// TIA Portal V19 export
FUNCTION_BLOCK "LMG7ApcFr_Std"   // FB19206, LAD
{ S7_Optimized_Access := 'TRUE' }
// stored: AutoNumber false, MemoryReserve 100, SetENOAutomatically false
   VAR_INPUT
      FirstCycle : Bool;
      InterlockGeneral : Bool := TRUE;
      Reset : Bool;
      StepNumberStarted : Int := 2;
      Frequency_1s : Bool;
      DebugMode : Bool;
      ActualTime : Time_Of_Day;
   END_VAR
   VAR_OUTPUT
      ActiveStep : Int;
      StateStopped : Bool;
      StateStarting : Bool;
      StateStarted : Bool;
      StateStopping : Bool;
      StateError : Bool;
      State : Int;
      StepError : Int;
      HistoricBuffer : Struct
         Index : Int := 0;
         BufferDetail : Array[0..9] of Struct
            TimeStartStep : Time_Of_Day;
            StepNumber : Int;
            ElapseTime_s : Int;
         END_STRUCT;
      END_STRUCT;
   END_VAR
   VAR_IN_OUT
      StepRequested : Int;
      StepTimeOut : Int;
   END_VAR
   VAR
      statFrequency_1sOld : Bool;
      statEdgeUpFrequency_1s : Bool;
   END_VAR
   VAR RETAIN
      statStepRequested : Int;
      statCounterTimeOut : Int;
      StatHistoricBuffer : Struct
         Index : Int := 0;
         BufferDetail : Array[0..9] of Struct
            TimeStartStep : Time_Of_Day;
            StepNumber : Int;
            ElapseTime_s : Int;
         END_STRUCT;
      END_STRUCT;
   END_VAR
   VAR
      instF_TRIG_StepStopped { S7_SetPoint := 'True'} : F_TRIG;
      instF_TRIG_StepStarted { S7_SetPoint := 'True'} : F_TRIG;
   END_VAR
BEGIN

REGION Network 1 (SCL): (*** COMMENTS ***)
   //=============================================================================
   //SIEMENS AG
   //(c)Copyright 2016 All Rights Reserved
   //-----------------------------------------------------------------------------
   //Requirements:
   //Functionality: G7 management of step
   //               Hystoric buffer of 10 entries. Need egde of 1s and time of the PLC
   //Supported types:
   //-----------------------------------------------------------------------------
   //Change log table:
   //Version       Date            Expert in charge    Changes applied
   //01.01.00      09.04.2020      PdA                 First release
   //01.02.00      01.07.2021      PdA                 TimeOut management
   //                                                  New organization 
   //01.03.00      19.03.2024      PdA                 Replace Enable by FirstCycle
   //                                                  Delete InterlockStartUp parameters
   //=============================================================================
END_REGION

REGION Network 2 (SCL): First call
   IF #FirstCycle THEN
       #StateStopped := TRUE;
       #StateStarting := FALSE;
       #StateStarted := FALSE;
       #StateStopping := FALSE;
       #ActiveStep := 0;
       #StepTimeOut := 0;
       #StepRequested := 0;
       #StepError := 0;
       #statStepRequested := 0;
       #statCounterTimeOut := 0;
   END_IF;
END_REGION

REGION Network 3 (SCL): Step Requested
   IF NOT #StateError THEN
       IF NOT #InterlockGeneral THEN
           #statStepRequested := 0;
           #StepRequested := 0;
       ELSIF (#statCounterTimeOut > #StepTimeOut) THEN
           #statStepRequested := "LMAG7_STEP_NUMBER_ERROR";
           #StepError := #ActiveStep;
       ELSE
           #statStepRequested := #StepRequested;
       END_IF;
   ELSE
       IF #Reset THEN
           #statStepRequested := 0;
           #StepError := 0;
       END_IF;
   END_IF;

   IF (#statStepRequested <> #ActiveStep) THEN
       #ActiveStep := #statStepRequested;
       #StepRequested := #statStepRequested;

       #StatHistoricBuffer.Index := #StatHistoricBuffer.Index + 1;
       IF #StatHistoricBuffer.Index > 9 THEN
           #StatHistoricBuffer.Index := 0;
       END_IF;
       #StatHistoricBuffer.BufferDetail[#StatHistoricBuffer.Index].TimeStartStep := #ActualTime;
       #StatHistoricBuffer.BufferDetail[#StatHistoricBuffer.Index].StepNumber := #statStepRequested;
       #StatHistoricBuffer.BufferDetail[#StatHistoricBuffer.Index].ElapseTime_s := #statCounterTimeOut;

       #statCounterTimeOut := 0;
       #StepTimeOut := 0;

   END_IF;

   #statEdgeUpFrequency_1s := #Frequency_1s AND NOT #statFrequency_1sOld;
   #statFrequency_1sOld := #Frequency_1s;

   IF (#StepTimeOut > 0) AND #statEdgeUpFrequency_1s AND NOT #DebugMode THEN
       #statCounterTimeOut := #statCounterTimeOut + 1;
   END_IF;

   #ActiveStep := #statStepRequested;
END_REGION

REGION Network 4: Output State Stopped, Started, Error
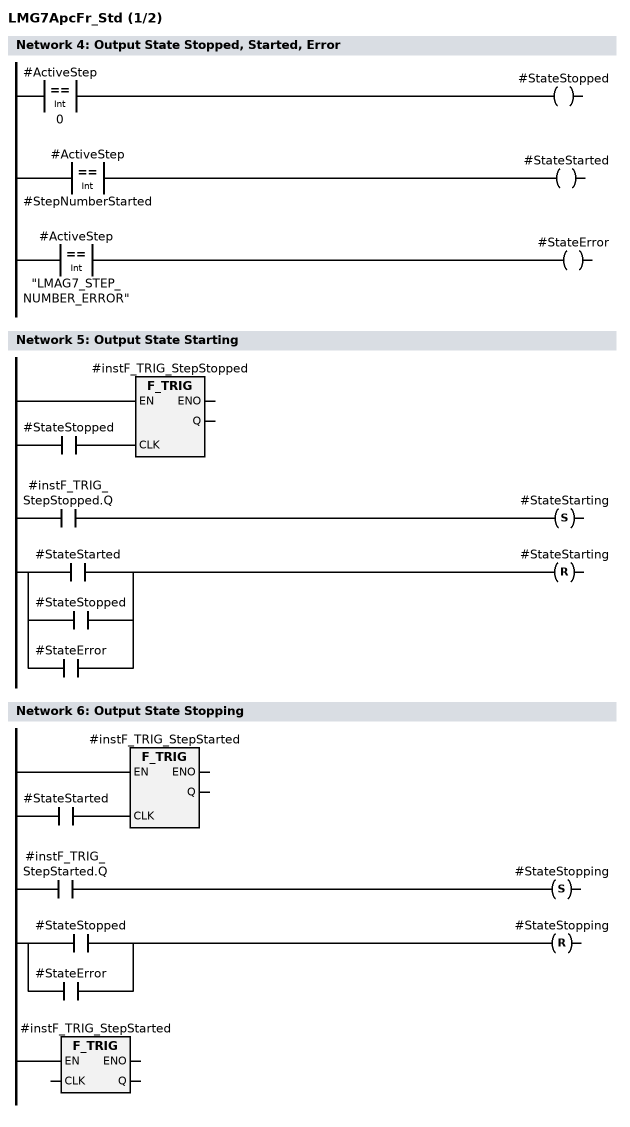
   RUNG wire#powerrail
      { S7_Templates := "SrcType := Int" } EQ_Contact(in1 := #ActiveStep, in2 := 0)
      Coil( #StateStopped )
   END_RUNG
   RUNG wire#powerrail
      { S7_Templates := "SrcType := Int" } EQ_Contact(in1 := #ActiveStep, in2 := #StepNumberStarted)
      Coil( #StateStarted )
   END_RUNG
   RUNG wire#powerrail
      { S7_Templates := "SrcType := Int" } EQ_Contact(in1 := #ActiveStep, in2 := "LMAG7_STEP_NUMBER_ERROR")
      Coil( #StateError )
   END_RUNG
   // the same network as SCL:
   #StateStopped := #ActiveStep = 0;
   #StateStarted := #ActiveStep = #StepNumberStarted;
   #StateError := #ActiveStep = "LMAG7_STEP_NUMBER_ERROR";
END_REGION

REGION Network 5: Output State Starting
   RUNG wire#powerrail
      #instF_TRIG_StepStopped.F_TRIG(CLK := wire#w1, Q =>)
   END_RUNG
   RUNG wire#powerrail
      Contact( #StateStopped )
   END_RUNG wire#w1
   RUNG wire#powerrail
      Contact( #instF_TRIG_StepStopped.Q )
      S_Coil( #StateStarting )
   END_RUNG
   RUNG wire#powerrail
      Contact( #StateStarted )
      wire#w2
      R_Coil( #StateStarting )
   END_RUNG
   RUNG wire#powerrail
      Contact( #StateStopped )
   END_RUNG wire#w2
   RUNG wire#powerrail
      Contact( #StateError )
   END_RUNG wire#w2
   // the same network as SCL:
   #instF_TRIG_StepStopped(CLK := #StateStopped);   // F_TRIG
   IF #instF_TRIG_StepStopped.Q THEN #StateStarting := TRUE; END_IF;
   IF #StateStarted OR #StateStopped OR #StateError THEN #StateStarting := FALSE; END_IF;
END_REGION

REGION Network 6: Output State Stopping
   RUNG wire#powerrail
      #instF_TRIG_StepStarted.F_TRIG(CLK := wire#w1, Q =>)
   END_RUNG
   RUNG wire#powerrail
      Contact( #StateStarted )
   END_RUNG wire#w1
   RUNG wire#powerrail
      Contact( #instF_TRIG_StepStarted.Q )
      S_Coil( #StateStopping )
   END_RUNG
   RUNG wire#powerrail
      Contact( #StateStopped )
      wire#w2
      R_Coil( #StateStopping )
   END_RUNG
   RUNG wire#powerrail
      Contact( #StateError )
   END_RUNG wire#w2
   RUNG wire#powerrail
      #instF_TRIG_StepStarted.F_TRIG(CLK :=, Q =>)
   END_RUNG
   // the same network as SCL:
   #instF_TRIG_StepStarted(CLK := #StateStarted);   // F_TRIG
   IF #instF_TRIG_StepStarted.Q THEN #StateStopping := TRUE; END_IF;
   IF #StateStopped OR #StateError THEN #StateStopping := FALSE; END_IF;
   #instF_TRIG_StepStarted();   // F_TRIG
END_REGION

REGION Network 7: Output State G7
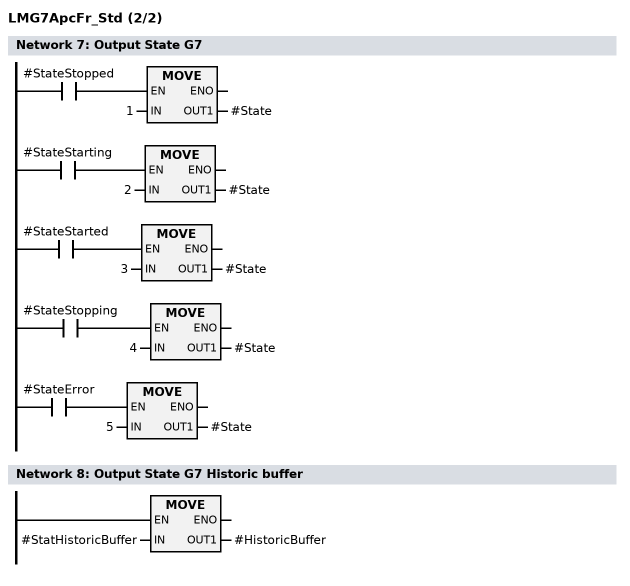
   RUNG wire#powerrail
      Contact( #StateStopped )
      Move(in := 1, out1 => #State)
   END_RUNG
   RUNG wire#powerrail
      Contact( #StateStarting )
      Move(in := 2, out1 => #State)
   END_RUNG
   RUNG wire#powerrail
      Contact( #StateStarted )
      Move(in := 3, out1 => #State)
   END_RUNG
   RUNG wire#powerrail
      Contact( #StateStopping )
      Move(in := 4, out1 => #State)
   END_RUNG
   RUNG wire#powerrail
      Contact( #StateError )
      Move(in := 5, out1 => #State)
   END_RUNG
   // the same network as SCL:
   IF #StateStopped THEN #State := 1; END_IF;
   IF #StateStarting THEN #State := 2; END_IF;
   IF #StateStarted THEN #State := 3; END_IF;
   IF #StateStopping THEN #State := 4; END_IF;
   IF #StateError THEN #State := 5; END_IF;
END_REGION

REGION Network 8: Output State G7 Historic buffer
   RUNG wire#powerrail
      Move(in := #StatHistoricBuffer, out1 => #HistoricBuffer)
   END_RUNG
   // the same network as SCL:
   #HistoricBuffer := #StatHistoricBuffer;
END_REGION
END_FUNCTION_BLOCK
